(* PLC project Unnamed, Unknown Unnamed 1 *)
(* stored: creationDateTime 2025-11-04T16:47:04, modificationDateTime 2025-11-04T16:50:06 *)

PROGRAM main
  VAR
    Trigger : BOOL := False;
    MemoryCoil : BOOL := False;
    BreakCondition : BOOL := False;
  END_VAR

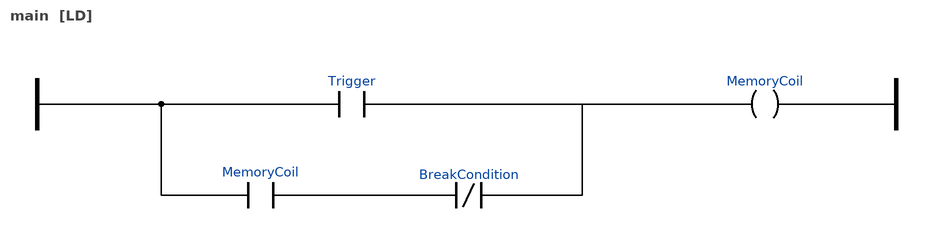
(* LD diagram, written out as Structured Text *)
MemoryCoil := Trigger OR MemoryCoil AND NOT BreakCondition;
END_PROGRAM

CONFIGURATION Config0
  RESOURCE Res0 ON PLC
    TASK task0(INTERVAL := T#20ms, PRIORITY := 0);
    PROGRAM instance0 WITH task0 : main;
  END_RESOURCE
END_CONFIGURATION
